TYPE ST_LoggedValues :
STRUCT
	nMotorFluxVoltage : INT;
END_STRUCT
END_TYPE

(* stored: Version 1.1.0.1, ProductVersion 3.1.4020.12
   DUT ST_LoggedValues: Id {97732bce-64c9-4020-bd74-d4a942b13940} *)
